# EPICS substitutions: iocs/example/exampleApp/Db/example_expanded.substitutions
# This file was automatically generated on Fri 28 Oct 2022 11:33:07 BST from
# source: /dls_sw/work/common/hir12111/support/amc100/etc/makeIocs/example.xml
#
# *** Please do not edit this file: edit the source file instead. ***
#

# Macros:
#  P     PV names Prefix (for motor record)
#  R     PV Name R component (for motor record)
#  name  Identifier for this motor instance
file $(AMC100)/db/AMC100Controller.template
{
pattern { P, R, PORT, TIMEOUT, name }
    { "AMC100TEST", ":CNTL", "AMC100TS.CNTL", "1", "AMC100TS.CNTL" }
}

# Macros:
#  P     PV names Prefix (for motor record)
#  R     PV Name R component (for motor record)
#  name  Name for entry
file $(AMC100)/db/AMC100Axis.template
{
pattern { P, R, PORT, AXIS, TIMEOUT, name }
    { "AMC100TEST", ":AX0", "AMC100TS.CNTL", "0", "3", "AMC100TS.AX1" }
    { "AMC100TEST", ":AX1", "AMC100TS.CNTL", "1", "3", "AMC100TS.AX2" }
}

# Macros:
#  P           Device Prefix
#  M           Device Suffix
#  PORT        Asyn port for motor record
#  ADDR        Address on controller
#  DESC        Description, displayed on EDM screen
#  MRES        Motor Step Size (EGU)
#  VELO        Velocity (EGU/s)
#  PREC        Display Precision
#  EGU         Engineering Units
#  TWV         Tweak Step Size (EGU)
#  DTYP        DTYP of record
#  DIR         User Direction
#  VBAS        Base Velocity (EGU/s)
#  VMAX        Max Velocity (EGU/s), defaults to VELO
#  ACCL        Seconds to Velocity
#  BDST        BL Distance (EGU)
#  BVEL        BL Velocity (EGU/s)
#  BACC        BL Seconds to Veloc.
#  DHLM        Dial High Limit
#  DLLM        Dial Low Limit
#  HLM         User High Limit
#  LLM         User Low Limit
#  HLSV        HW Lim. Violation Svr
#  INIT        Startup commands
#  SREV        Steps per Revolution
#  RRES        Readback Step Size (EGU)
#  ERES        Encoder Step Size (EGU)
#  JAR         Jog Acceleration (EGU/s^2)
#  UEIP        Use Encoder If Present
#  URIP        Use RDBL If Present
#  RDBL        Readback Location, set URIP = 1 if you specify this
#  RLNK        Readback output link
#  RTRY        Max retry count
#  DLY         Readback settle time (s)
#  OFF         User Offset (EGU)
#  RDBD        Retry Deadband (EGU)
#  FOFF        Freeze Offset, 0=variable, 1=frozen
#  ADEL        Alarm monitor deadband (EGU)
#  NTM         New Target Monitor, only set to 0 for soft motors
#  FEHIGH      HIGH limit for following error
#  FEHIHI      HIHI limit for following error
#  FEHHSV      HIHI alarm severity for following error
#  FEHSV       HIGH alarm severity for following error
#  SCALE       Scale factor, if pmacSetAxisScale is used this should be set
#  HOMEVIS     If 1 then home is visible on the gui
#  HOMEVISSTR  If HOMEVIS=0, then display this text on the gui instead
#  name        Object name and gui association name
#  alh         Set this to alh to add the motor to the alarm handler and send emails,
#  gda_name    Name to export this as to GDA
#  gda_desc    Description to export this as to GDA
file $(MOTOR)/db/basic_asyn_motor.template
{
pattern { P, M, PORT, ADDR, DESC, MRES, VELO, PREC, EGU, TWV, DTYP, DIR, VBAS, VMAX, ACCL, BDST, BVEL, BACC, DHLM, DLLM, HLM, LLM, HLSV, INIT, SREV, RRES, ERES, JAR, UEIP, URIP, RDBL, RLNK, RTRY, DLY, OFF, RDBD, FOFF, ADEL, NTM, FEHIGH, FEHIHI, FEHHSV, FEHSV, SCALE, HOMEVIS, HOMEVISSTR, name, alh, gda_name, gda_desc }
    { "AMC100TEST", ":X", "AMC100TS.CNTL", "0", "Axis X", "0.001", "2", "3", "um", "5", "asynMotor", "0", "0", "$(VELO)", "0.5", "0", "0", "", "10000", "-10000", "", "", "MAJOR", "", "1000", "", "", "", "0", "0", "", "", "0", "0", "0", "", "0", "0", "1", "0", "0", "NO_ALARM", "NO_ALARM", "1", "1", "Use motor summary screen", "AMC100TS.M1", "None", "", "$(DESC)" }
    { "AMC100TEST", ":Y", "AMC100TS.CNTL", "1", "Axis Y", "0.001", "2", "3", "um", "5", "asynMotor", "0", "0", "$(VELO)", "0.5", "0", "0", "", "10000", "-10000", "", "", "MAJOR", "", "1000", "", "", "", "0", "0", "", "", "0", "0", "0", "", "0", "0", "1", "0", "0", "NO_ALARM", "NO_ALARM", "1", "1", "Use motor summary screen", "AMC100TS.M2", "None", "", "$(DESC)" }
}
